// TIA Portal V20 export
DATA_BLOCK "InstCallEquipment"   // DB139
{ DB_Accessible_From_OPC_UA := 'FALSE' }
AUTHOR : ERsystem_FA2_DH. Kim
// stored: AssignedProDiagFB Unit1.Em1.ProDiag, DBAccessibleFromOPCUA false, DBAccessibleFromWebserver false, InstanceOfName Unit1.Em1.CallEquipment, InstanceOfType FB, Namespace Unit1.Em1
"Unit1.Em1.CallEquipment"
   // VAR_INPUT
   //    ZoneOperationEnable { ExternalWritable := 'False'} : "LWONIK_typeSafetyZoneManualOperation";
   // END_VAR
   // VAR_IN_OUT
   //    unitStatus : "LAF_typeUnitStatus";
   //    unitAlarmDB : "LAF_typeAlarms";
   //    emFeedback : "LUC_typeEmFeedback";
   // END_VAR
   // VAR
   //    instSequenceUnwinder { S7_SetPoint := 'True'} : "Unit1.Em1.Sequence_1_SepaUnwinderBtm";
   //    instBtmHomeJob1 { S7_SetPoint := 'True'} : "LAF_SelectJob";
   //    instBtmRewidnigJob10 { S7_SetPoint := 'True'} : "LAF_SelectJob";
   //    instBtmUnwindingJob2 { S7_SetPoint := 'True'} : "LAF_SelectJob";
   //    instBtmStopJob3 { S7_SetPoint := 'True'} : "LAF_SelectJob";
   //    instBtmRewidnigJob4 { S7_SetPoint := 'True'} : "LAF_SelectJob";
   //    instCmBtmDirectionCheckSensor { S7_SetPoint := 'True'} : "LBC_DigitalSignalCn";
   //    instCmUnwinderBottomRadiusMeasure { ExternalAccessible := 'False'; ExternalVisible := 'False'; ExternalWritable := 'False'} : "LBC_AnalogInputCn";
   //    instCmRadiusMeasure { S7_SetPoint := 'True'} : "LER_RadiusMeasure";
   //    instCmUnwinderBottomAxisB { S7_SetPoint := 'True'} : "LBC_Axis64Pos_TecPlcCn";
   //    instInterlockCmUnwinderBtmAxisB { S7_SetPoint := 'True'} : "LER_Axis64Pos_InterlockSummary";
   //    instCmUnwinderAirShaftBottomOnOff { ExternalAccessible := 'False'; ExternalVisible := 'False'; ExternalWritable := 'False'; S7_SetPoint := 'True'} : "LBC_TwoWayActuatorCn";
   //    instCmUnwinderBottomEpcControllerInterface { ExternalAccessible := 'False'; ExternalVisible := 'False'; ExternalWritable := 'False'; S7_SetPoint := 'True'} : "LER_EPC_CON600";
   //    instManageAlarms { ExternalWritable := 'False'} : "LAF_ManageAlarms";
   //    instEventsPFE : "Unit1.Em1.EventsPFE";
   //    instLER_BrakeTestUnwinderBottomAxisB : "LER_BrakeTest";
   //    statUnitStatus { ExternalWritable := 'False'} : "LAF_typeUnitStatus";
   //    statSlmStatus : Struct
   //       running { ExternalWritable := 'False'} : Bool;
   //       powerOff { ExternalWritable := 'False'} : Bool;
   //    END_STRUCT;
   //    statAllBrakeTest { ExternalWritable := 'False'} : "LER_typeBrakeTestUnitCommands";
   //    statTonTime { ExternalAccessible := 'False'; ExternalVisible := 'False'; ExternalWritable := 'False'} : Array[0..1999] of TON_TIME;
   //    statTofTime { ExternalAccessible := 'False'; ExternalVisible := 'False'; ExternalWritable := 'False'} : Array[0..99] of TOF_TIME;
   //    statPulse { ExternalAccessible := 'False'; ExternalVisible := 'False'; ExternalWritable := 'False'} : Struct
   //       miscellaneous : Array[0..99] of Bool;
   //       workingDone : Struct
   //          mainPnP : Array[0..99] of Bool;
   //          alignTable : Array[0..99] of Bool;
   //          ngPnP : Array[0..99] of Bool;
   //       END_STRUCT;
   //       axisEnable : Array[0..99] of Bool;
   //       brakeTest : Array[0..99] of Bool;
   //    END_STRUCT;
   //    statEnableManualCmds : Bool := TRUE;
   //    statRcEnableCmds : Bool;
   //    Scan_on : Bool;
   //    "*** Interlock Axis ***" { ExternalAccessible := 'False'; ExternalVisible := 'False'; ExternalWritable := 'False'} : Bool;
   //    "UnwinderBtmAxisB Home" { S7_SetPoint := 'True'} : "Homing.LER_Axis";
   //    "UnwinderBtmAxisB Jog_CW" { S7_SetPoint := 'True'} : "Jog.LER_Axis";
   //    "UnwinderBtmAxisB Jog_CCW" { S7_SetPoint := 'True'} : "Jog.LER_Axis";
   //    "UnwinderBtmAxisB Position" { S7_SetPoint := 'True'} : Array[0..5] of "Position.LER_Axis";
   //    "*** Interlock Actuator ******" { ExternalAccessible := 'False'; ExternalVisible := 'False'; ExternalWritable := 'False'; S7_SetPoint := 'True'} : Bool;
   //    "UnwinderAirShaftBottom On" { S7_SetPoint := 'True'} : "Cylinder.LER_Actuator";
   //    "UnwinderAirShaftBottom Off" { S7_SetPoint := 'True'} : "Cylinder.LER_Actuator";
   //    AXIS2 : "LER_CM_Name";
   //    Cylinder2 : "LER_CM_Name";
   //    citi_Ptrig : Array[0..20] of Bool;
   //    citiTon : Array[0..20] of TON_TIME;
   //    citi : Time;
   //    citiTest : Array[0..20] of Bool;
   // END_VAR
BEGIN
   ZoneOperationEnable.autoStartEnable := FALSE;
   ZoneOperationEnable.doorLockEnable := TRUE;
   ZoneOperationEnable.doorUnlockEnable := TRUE;
   ZoneOperationEnable.rc_AutoEnable := FALSE;
   ZoneOperationEnable.rc_RollChangeEnable := FALSE;
   ZoneOperationEnable.rc_DoorLockEnable := TRUE;
   ZoneOperationEnable.rc_DoorUnlockEnable := TRUE;
   ZoneOperationEnable.hmiOperationEnable := TRUE;
   ZoneOperationEnable.phmiOperationEnable := FALSE;
   instCmBtmDirectionCheckSensor.enable := TRUE;
   instCmBtmDirectionCheckSensor.parentReferenceDesignator := WSTRING#'U1.EM1 SepaUnwinderBtm';
   instCmBtmDirectionCheckSensor.digitalValue := TRUE;
   instCmBtmDirectionCheckSensor.simulatedDigitalValue := FALSE;
   instCmBtmDirectionCheckSensor.statProcessValues.enable := TRUE;
   instCmBtmDirectionCheckSensor.statProcessValues.referenceDesignator := WSTRING#'U1.EM1 SepaUnwinderBtm.cmBtmDirectionCheckSensor';
   instCmBtmDirectionCheckSensor.statProcessValues.simulation := FALSE;
   instCmBtmDirectionCheckSensor.statProcessValues.processValue := TRUE;
   instCmBtmDirectionCheckSensor.statProcessValues.error := FALSE;
   instCmBtmDirectionCheckSensor.statProcessValues.status := 16#0000;
   instCmBtmDirectionCheckSensor.statDiagnostics.status := 16#0000;
   instCmBtmDirectionCheckSensor.statDiagnostics.subfunctionStatus := 16#0000;
   instCmBtmDirectionCheckSensor.statDiagnostics.stateNumber := 0;
   instCmBtmDirectionCheckSensor.statEmptyDiagnostics.status := 16#0000;
   instCmBtmDirectionCheckSensor.statEmptyDiagnostics.subfunctionStatus := 16#0000;
   instCmBtmDirectionCheckSensor.statEmptyDiagnostics.stateNumber := 0;
   instCmBtmDirectionCheckSensor.instOnDelay.PT := T#0MS;
   instCmBtmDirectionCheckSensor.instOnDelay.IN := FALSE;
   instCmBtmDirectionCheckSensor.instOffDelay.PT := T#0MS;
   instCmBtmDirectionCheckSensor.instOffDelay.IN := FALSE;
   instCmBtmDirectionCheckSensor.statDisableAlarms := FALSE;
   instCmBtmDirectionCheckSensor.statErrorState := 16#0000;
   instCmBtmDirectionCheckSensor.statFirstCall := FALSE;
   instCmBtmDirectionCheckSensor.statResetPrevious := FALSE;
   instCmBtmDirectionCheckSensor.statEnablePrevious := TRUE;
   instCmBtmDirectionCheckSensor.statProcessValuePrevious := TRUE;
   instCmUnwinderBottomRadiusMeasure.enable := TRUE;
   instCmUnwinderBottomRadiusMeasure.parentReferenceDesignator := WSTRING#'U1.EM1 SepaUnwinderBtm';
   instCmUnwinderBottomRadiusMeasure.analogValue := -32768;
   instCmUnwinderBottomRadiusMeasure.simulatedAnalogValue := 0;
   instCmUnwinderBottomRadiusMeasure.statProcessValues.enable := TRUE;
   instCmUnwinderBottomRadiusMeasure.statProcessValues.referenceDesignator := WSTRING#'U1.EM1 SepaUnwinderBtm.cmRadiusMeasureBtm';
   instCmUnwinderBottomRadiusMeasure.statProcessValues.simulation := FALSE;
   instCmUnwinderBottomRadiusMeasure.statProcessValues.processValue := 0.0;
   instCmUnwinderBottomRadiusMeasure.statProcessValues.analogValue := -4864;
   instCmUnwinderBottomRadiusMeasure.statProcessValues.limitHigh2 := FALSE;
   instCmUnwinderBottomRadiusMeasure.statProcessValues.limitHigh1 := FALSE;
   instCmUnwinderBottomRadiusMeasure.statProcessValues.limitLow1 := TRUE;
   instCmUnwinderBottomRadiusMeasure.statProcessValues.limitLow2 := TRUE;
   instCmUnwinderBottomRadiusMeasure.statProcessValues.maxValueReached := FALSE;
   instCmUnwinderBottomRadiusMeasure.statProcessValues.minValueReached := TRUE;
   instCmUnwinderBottomRadiusMeasure.statProcessValues.error := TRUE;
   instCmUnwinderBottomRadiusMeasure.statProcessValues.status := 16#8405;
   instCmUnwinderBottomRadiusMeasure.statDiagnostics.status := 16#8405;
   instCmUnwinderBottomRadiusMeasure.statDiagnostics.subfunctionStatus := 16#0000;
   instCmUnwinderBottomRadiusMeasure.statDiagnostics.stateNumber := 0;
   instCmUnwinderBottomRadiusMeasure.statEmptyDiagnostics.status := 16#0000;
   instCmUnwinderBottomRadiusMeasure.statEmptyDiagnostics.subfunctionStatus := 16#0000;
   instCmUnwinderBottomRadiusMeasure.statEmptyDiagnostics.stateNumber := 0;
   instCmUnwinderBottomRadiusMeasure.statLimitationMessage := '-70.37 unit < 0.00 unit';
   instCmUnwinderBottomRadiusMeasure.statLimitMessage := '0.00 unit <= 0.00 unit';
   instCmUnwinderBottomRadiusMeasure.statErrorState := 16#8405;
   instCmUnwinderBottomRadiusMeasure.statFirstCall := FALSE;
   instCmUnwinderBottomRadiusMeasure.statDisableAlarms := TRUE;
   instCmUnwinderBottomRadiusMeasure.statResetPrevious := FALSE;
   instCmUnwinderBottomRadiusMeasure.statEnablePrevious := TRUE;
   instCmUnwinderAirShaftBottomOnOff.enable := TRUE;
   instCmUnwinderAirShaftBottomOnOff.parentReferenceDesignator := WSTRING#'U1.EM1 SepaUnwinderBtm';
   instCmUnwinderAirShaftBottomOnOff.feedbackHomePos := FALSE;
   instCmUnwinderAirShaftBottomOnOff.feedbackWorkPos := FALSE;
   instCmUnwinderAirShaftBottomOnOff.enableManualCmds := TRUE;
   instCmUnwinderAirShaftBottomOnOff.interlockWorkPos := TRUE;
   instCmUnwinderAirShaftBottomOnOff.interlockHomePos := TRUE;
   instCmUnwinderAirShaftBottomOnOff.goToHomePos := FALSE;
   instCmUnwinderAirShaftBottomOnOff.goToWorkPos := FALSE;
   instCmUnwinderAirShaftBottomOnOff.statProcessValues.enable := TRUE;
   instCmUnwinderAirShaftBottomOnOff.statProcessValues.referenceDesignator := WSTRING#'U1.EM1 SepaUnwinderBtm.cmAirShaftBtmOnOff';
   instCmUnwinderAirShaftBottomOnOff.statProcessValues.commandHomePos := FALSE;
   instCmUnwinderAirShaftBottomOnOff.statProcessValues.commandWorkPos := FALSE;
   instCmUnwinderAirShaftBottomOnOff.statProcessValues.goToHomePos := FALSE;
   instCmUnwinderAirShaftBottomOnOff.statProcessValues.goToWorkPos := FALSE;
   instCmUnwinderAirShaftBottomOnOff.statProcessValues.inHomePos := FALSE;
   instCmUnwinderAirShaftBottomOnOff.statProcessValues.inWorkPos := FALSE;
   instCmUnwinderAirShaftBottomOnOff.statProcessValues.reset := FALSE;
   instCmUnwinderAirShaftBottomOnOff.statProcessValues.enableManualCmds := TRUE;
   instCmUnwinderAirShaftBottomOnOff.statProcessValues.error := FALSE;
   instCmUnwinderAirShaftBottomOnOff.statProcessValues.interlockHomePos := TRUE;
   instCmUnwinderAirShaftBottomOnOff.statProcessValues.interlockWorkPos := TRUE;
   instCmUnwinderAirShaftBottomOnOff.statProcessValues.status := 16#7003;
   instCmUnwinderAirShaftBottomOnOff.statProcessValues.interlockWarningWorkPos := FALSE;
   instCmUnwinderAirShaftBottomOnOff.statProcessValues.interlockWarningHomePos := FALSE;
   instCmUnwinderAirShaftBottomOnOff.statCurrentInputs.commandHomePos := FALSE;
   instCmUnwinderAirShaftBottomOnOff.statCurrentInputs.commandWorkPos := FALSE;
   instCmUnwinderAirShaftBottomOnOff.statCurrentInputs.reset := FALSE;
   instCmUnwinderAirShaftBottomOnOff.statPreviousInputs.commandHomePos := FALSE;
   instCmUnwinderAirShaftBottomOnOff.statPreviousInputs.commandWorkPos := FALSE;
   instCmUnwinderAirShaftBottomOnOff.statPreviousInputs.reset := FALSE;
   instCmUnwinderAirShaftBottomOnOff.statCurrentInterface.commandHomePos := FALSE;
   instCmUnwinderAirShaftBottomOnOff.statCurrentInterface.commandWorkPos := FALSE;
   instCmUnwinderAirShaftBottomOnOff.statCurrentInterface.reset := FALSE;
   instCmUnwinderAirShaftBottomOnOff.statPreviousInterface.commandHomePos := FALSE;
   instCmUnwinderAirShaftBottomOnOff.statPreviousInterface.commandWorkPos := FALSE;
   instCmUnwinderAirShaftBottomOnOff.statPreviousInterface.reset := FALSE;
   instCmUnwinderAirShaftBottomOnOff.statEmptyDiagnostics.status := 16#0000;
   instCmUnwinderAirShaftBottomOnOff.statEmptyDiagnostics.subfunctionStatus := 16#0000;
   instCmUnwinderAirShaftBottomOnOff.statEmptyDiagnostics.stateNumber := 0;
   instCmUnwinderAirShaftBottomOnOff.instTimerReachPos.PT := T#0MS;
   instCmUnwinderAirShaftBottomOnOff.instTimerReachPos.IN := FALSE;
   instCmUnwinderAirShaftBottomOnOff.instTimerLeavePos.PT := T#0MS;
   instCmUnwinderAirShaftBottomOnOff.instTimerLeavePos.IN := FALSE;
   instCmUnwinderAirShaftBottomOnOff.instTimerDiscrepancyCheck.PT := T#0MS;
   instCmUnwinderAirShaftBottomOnOff.instTimerDiscrepancyCheck.IN := FALSE;
   instCmUnwinderAirShaftBottomOnOff.statDisableAlarms := FALSE;
   instCmUnwinderAirShaftBottomOnOff.statDiagnostics.status := 16#7003;
   instCmUnwinderAirShaftBottomOnOff.statDiagnostics.subfunctionStatus := 16#0000;
   instCmUnwinderAirShaftBottomOnOff.statDiagnostics.stateNumber := 0;
   instCmUnwinderAirShaftBottomOnOff.statEnablePrevious := TRUE;
   instCmUnwinderAirShaftBottomOnOff.statFirstCall := FALSE;
   instCmUnwinderAirShaftBottomOnOff.statResetPrevious := FALSE;
   instCmUnwinderAirShaftBottomOnOff.statValid := TRUE;
   instCmUnwinderAirShaftBottomOnOff.statBusy := TRUE;
   instCmUnwinderAirShaftBottomOnOff.statError := FALSE;
   instCmUnwinderAirShaftBottomOnOff.statInterlockWorkOff := FALSE;
   instCmUnwinderAirShaftBottomOnOff.statInterlockHomeOff := FALSE;
   instCmUnwinderAirShaftBottomOnOff.statFbState := 50;
   instCmUnwinderAirShaftBottomOnOff.statFbStatePrevious := 50;
   instCmUnwinderAirShaftBottomOnOff.statErrorUserCleared := FALSE;
   instCmUnwinderAirShaftBottomOnOff.statErrorAutoCleared := FALSE;
   instCmUnwinderAirShaftBottomOnOff.statErrorState := 16#0000;
   instCmUnwinderAirShaftBottomOnOff.statDisablingCompleted := FALSE;
   instCmUnwinderAirShaftBottomOnOff.statFeedbackHomePos := FALSE;
   instCmUnwinderAirShaftBottomOnOff.statFeedbackWorkPos := FALSE;
   instManageAlarms.proDiagState.Total_Number := 426;
   instManageAlarms.proDiagState.All := TRUE;
   instManageAlarms.proDiagState.O := FALSE;
   instManageAlarms.proDiagState.I := FALSE;
   instManageAlarms.proDiagState.R := FALSE;
   instManageAlarms.proDiagState."A" := FALSE;
   instManageAlarms.proDiagState.P := FALSE;
   instManageAlarms.proDiagState.Merr := TRUE;
   instManageAlarms.proDiagState.Mtxt := FALSE;
   instManageAlarms.proDiagState.SV_Types := 16#20;
   instManageAlarms.proDiagState.C1 := TRUE;
   instManageAlarms.proDiagState.C2 := FALSE;
   instManageAlarms.proDiagState.C3 := FALSE;
   instManageAlarms.proDiagState.C4 := FALSE;
   instManageAlarms.proDiagState.C5 := FALSE;
   instManageAlarms.proDiagState.C6 := FALSE;
   instManageAlarms.proDiagState.C7 := FALSE;
   instManageAlarms.proDiagState.C8 := FALSE;
   instManageAlarms.proDiagState.Categories := 16#01;
   instManageAlarms.proDiagState.Sub_Cat_1 := 16#0000_0001;
   instManageAlarms.proDiagState.Sub_Cat_2 := 16#0000_0000;
   instManageAlarms.proDiagState.Reserved := 16#00;
   instManageAlarms.parentAlarmDB.error := TRUE;
   instManageAlarms.parentAlarmDB.warning := FALSE;
   instManageAlarms.parentAlarmDB.info := FALSE;
   instManageAlarms.alarmDB.error := TRUE;
   instManageAlarms.alarmDB.warning := FALSE;
   instManageAlarms.alarmDB.info := FALSE;
   instManageAlarms.hmiInterfaceDB.error := TRUE;
   instManageAlarms.hmiInterfaceDB.warning := FALSE;
   instManageAlarms.hmiInterfaceDB.info := FALSE;
   statUnitStatus.acknowledgeActive := FALSE;
   statUnitStatus.alarmsDisabled := FALSE;
   statUnitStatus.simulationActive := FALSE;
   statUnitStatus.safetyReleased := TRUE;
   statUnitStatus.state.current := 2;
   statUnitStatus.state.clearing := FALSE;
   statUnitStatus.state.stopped := TRUE;
   statUnitStatus.state.starting := FALSE;
   statUnitStatus.state.idle := FALSE;
   statUnitStatus.state.suspended := FALSE;
   statUnitStatus.state.execute := FALSE;
   statUnitStatus.state.stopping := FALSE;
   statUnitStatus.state.aborting := FALSE;
   statUnitStatus.state.aborted := FALSE;
   statUnitStatus.state.holding := FALSE;
   statUnitStatus.state.held := FALSE;
   statUnitStatus.state.unholding := FALSE;
   statUnitStatus.state.suspending := FALSE;
   statUnitStatus.state.unsuspending := FALSE;
   statUnitStatus.state.resetting := FALSE;
   statUnitStatus.state.completing := FALSE;
   statUnitStatus.state.complete := FALSE;
END_DATA_BLOCK
